Staubli VAL3: ros_server.dtx

public JointFbkMsg rosJointFbkMsg
  [0]
    Body body
      [0]
        num nData[132]
    Header header
      [0]
        num nCommType = 1
        num nData[12]
        num nMsgType = 15
        num nReplyCode
    JointFeedback jointFeedback
      [0]
        num nAccelerations[10]
        num nPositions[10]
        num nRobotId
        num nTime
        num nValidFields
        num nVelocities[10]
    Prefix prefix
      [0]
        num nData[4]
        num nLength = 144
public JointStateMsg rosJointMsg
  [0]
    Body body
      [0]
        num nData[44]
    Header header
      [0]
        num nCommType = 1
        num nData[12]
        num nMsgType = 10
        num nReplyCode
    JointState jointState
      [0]
        num nJoints[10]
        num nSeq
    Prefix prefix
      [0]
        num nData[4]
        num nLength = 56
public JointTrajPtFMsg rosTrajPtFAck
  [0]
    Body body
      [0]
        num nData[136]
    Header header
      [0]
        num nCommType = 3
        num nData[12]
        num nMsgType = 14
        num nReplyCode = 1
    JointTrajPtFull jointTrajPtFull
      [0]
        num nAccelerations[10]
        num nPositions[10]
        num nRobotId
        num nSeq
        num nTime
        num nValidFields
        num nVelocities[10]
    Prefix prefix
      [0]
        num nData[4]
        num nLength = 148
public JointTrajPtFMsg rosTrajPtFMsg
  [0]
    Body body
      [0]
        num nData[136]
    Header header
      [0]
        num nCommType
        num nData[12]
        num nMsgType
        num nReplyCode
    JointTrajPtFull jointTrajPtFull
      [0]
        num nAccelerations[10]
        num nPositions[10]
        num nRobotId
        num nSeq
        num nTime
        num nValidFields
        num nVelocities[10]
    Prefix prefix
      [0]
        num nData[4]
        num nLength = 148
public JointTrajPtMsg rosTrajPtAck
  [0]
    Body body
      [0]
        num nData[52]
    Header header
      [0]
        num nCommType = 3
        num nData[12]
        num nMsgType = 11
        num nReplyCode = 1
    JointTrajPt jointTrajPt
      [0]
        num nDuration
        num nJoints[10]
        num nSeq
        num nVelocity
    Prefix prefix
      [0]
        num nData[4]
        num nLength = 64
public JointTrajPtMsg rosTrajPtMsg
  [0]
    Body body
      [0]
        num nData[52]
    Header header
      [0]
        num nCommType
        num nData[12]
        num nMsgType
        num nReplyCode
    JointTrajPt jointTrajPt
      [0]
        num nDuration
        num nJoints[10]
        num nSeq
        num nVelocity
    Prefix prefix
      [0]
        num nData[4]
        num nLength = 64
MotionCfgVel motionCfgVel
  [0]
    frame fReference = {fatherId=world[0]}
    mdesc mMaxSpeed = {leave=1, reach=1, blend=off}
    num nCmdType
    tool tTool = {fatherId=flange[0], ioLink=valve1}
MotionCmdVel motionCmdVel
  [0]
    num nCmdType
    num nSequence
    num nVelCmd[6]
MotionCmdVel actMotionCmdVel
  [0]
    num nCmdType
    num nSequence
    num nVelCmd[6]
public Queue qMoveBuffer
  [0]
    MotionCmd buffer[10]
      [0]
        jointRx jJointRx
        mdesc mDesc = {leave=0, reach=0}
        num nDuration
        num nSequence
      [1]
        jointRx jJointRx
        mdesc mDesc = {leave=0, reach=0}
        num nDuration
        num nSequence
      [2]
        jointRx jJointRx
        mdesc mDesc = {leave=0, reach=0}
        num nDuration
        num nSequence
      [3]
        jointRx jJointRx
        mdesc mDesc = {leave=0, reach=0}
        num nDuration
        num nSequence
      [4]
        jointRx jJointRx
        mdesc mDesc = {leave=0, reach=0}
        num nDuration
        num nSequence
      [5]
        jointRx jJointRx
        mdesc mDesc = {leave=0, reach=0}
        num nDuration
        num nSequence
      [6]
        jointRx jJointRx
        mdesc mDesc = {leave=0, reach=0}
        num nDuration
        num nSequence
      [7]
        jointRx jJointRx
        mdesc mDesc = {leave=0, reach=0}
        num nDuration
        num nSequence
      [8]
        jointRx jJointRx
        mdesc mDesc = {leave=0, reach=0}
        num nDuration
        num nSequence
      [9]
        jointRx jJointRx
        mdesc mDesc = {leave=0, reach=0}
        num nDuration
        num nSequence
    num nElems
    num nPop
    num nPush
public Queue qTrajPtBuffer
  [0]
    MotionCmd buffer[10]
      [0]
        jointRx jJointRx
        mdesc mDesc = {leave=0, reach=0}
        num nDuration
        num nSequence
      [1]
        jointRx jJointRx
        mdesc mDesc = {leave=0, reach=0}
        num nDuration
        num nSequence
      [2]
        jointRx jJointRx
        mdesc mDesc = {leave=0, reach=0}
        num nDuration
        num nSequence
      [3]
        jointRx jJointRx
        mdesc mDesc = {leave=0, reach=0}
        num nDuration
        num nSequence
      [4]
        jointRx jJointRx
        mdesc mDesc = {leave=0, reach=0}
        num nDuration
        num nSequence
      [5]
        jointRx jJointRx
        mdesc mDesc = {leave=0, reach=0}
        num nDuration
        num nSequence
      [6]
        jointRx jJointRx
        mdesc mDesc = {leave=0, reach=0}
        num nDuration
        num nSequence
      [7]
        jointRx jJointRx
        mdesc mDesc = {leave=0, reach=0}
        num nDuration
        num nSequence
      [8]
        jointRx jJointRx
        mdesc mDesc = {leave=0, reach=0}
        num nDuration
        num nSequence
      [9]
        jointRx jJointRx
        mdesc mDesc = {leave=0, reach=0}
        num nDuration
        num nSequence
    num nElems
    num nPop
    num nPush
public RobotStatusMsg rosStatusMsg
  [0]
    Body body
      [0]
        num nData[32]
    Header header
      [0]
        num nCommType = 1
        num nData[12]
        num nMsgType = 13
        num nReplyCode
    Prefix prefix
      [0]
        num nData[4]
        num nLength = 40
    RobotStatus robotStatus
      [0]
        num nDrivesPowered
        num nEStopped
        num nErrorCode
        num nInError
        num nInMotion
        num nMode
        num nMotionPossible
        num nTrajectoryComplete
public RosSimpleMsg genericMotMsg
  [0]
    Header header
      [0]
        num nMsgType
        num nCommType
        num nReplyCode
        num nData[12]
    Prefix prefix
      [0]
        num nLength
        num nData[4]
public RosSimpleMsg genericSysMsg
  [0]
    Header header
      [0]
        num nMsgType
        num nCommType
        num nReplyCode
        num nData[12]
    Prefix prefix
      [0]
        num nLength
        num nData[4]
public RosSimpleMsg genericIOMsg
  [0]
    Header header
      [0]
        num nMsgType
        num nCommType
        num nReplyCode
        num nData[12]
    Prefix prefix
      [0]
        num nLength
        num nData[4]
public _MsgRecvState MsgRecvState
  [0]
    num DECODE_BODY
    num DECODE_HEADER
    num HANDLE_REQUEST
    num PUSH_MOTION
    num RECEIVE_BODY
    num RECEIVE_HEADER
    num SEND_ACK
public bool bDataIn
public bool bDataOut
public bool bDebugMode
public bool bFbkOverrun
public bool bMotionMsgEvent
public bool bMotionOverrun
public bool bOverwriteVel
public bool bRecvOverrun
public bool bScreenOverrun
public bool bShowDebug
public bool bStopNow
public num nConnFlagIO
public num nConnFlagMotion
public num nConnFlagState
public num nConnFlagSystem
public num nDebugCursor
public num nDebugLevel = 5
public num nDebugLevelMax = 7
public num nElapsedTime
public num nHeaderTime = 0.004
num nMotionMode = 1
public num nMotionMsgType
num nMotionPeriod = 0.004
public num nMotionProgress
public num nMoveId = -1
public num nMovePts
public num nPtsPopped
public sio siTcpIpIO = {link=Socket\IO}
public sio siTcpIpMotion = {link=Socket\Motion}
public sio siTcpIpState = {link=Socket\State}
public sio siTcpIpSystem = {link=Socket\System}
public string sHeartbeatTask = "htbtTask"
public string sIORequestTask = "ioRequestTask"
public string sMotionRecvTask = "motionRecvTask"
public string sMotionTask = "motionTask"
public string sScreenTask = "screenTask"
public string sStateMachTask = "stateTask"
public string sStreamerTask = "streamerTask"
public string sSysRequestTask
public tool tTool = {fatherId=flange[0], ioLink=valve1}
jointRx jPosition
jointRx jSpeed
num nTotalTrajPoint
